# EPICS autosave request: mcaApp/Db/mca_settings.req
# FILE... mca_settings.req
# USAGE.. mca.db fields autosave'd.
file "simple_mca_settings.req", P=$(P), M=$(M)
$(P)$(M)Read.SCAN
$(P)$(M)Status.SCAN
